FUNCTION_BLOCK PalletizerElevator EXTENDS Elevator
VAR_INPUT
END_VAR
VAR_OUTPUT
	isMoving : BOOL;
END_VAR
VAR
	fbElevatorMoving : Sensor;
	fbElevatorUp : BoolOut;
	fbElevatorDown : BoolOut;
	fbElevatorToLimit : BoolOut;
END_VAR

isMoving := fbElevatorMoving.bSignal;

PROPERTY getElevatorMoving : I_StepCondition
GET
getElevatorMoving := fbElevatorMoving.getSignal;
END_GET
END_PROPERTY

METHOD MoveDown : BOOL
VAR_INPUT
END_VAR
fbElevatorDown.setValue := TRUE;
fbElevatorUp.setValue := FALSE;

fbElevatorToLimit.setValue := TRUE;
END_METHOD

METHOD MoveUp : BOOL
VAR_INPUT
END_VAR
fbElevatorUp.setValue := TRUE;
fbElevatorDown.setValue := FALSE;

fbElevatorToLimit.setValue := TRUE;
END_METHOD

END_FUNCTION_BLOCK

(* stored: Version 1.1.0.1, ProductVersion 3.1.4024.2
   POU PalletizerElevator: Id {4eb779f8-64c2-45d2-8e33-ff6a6414ef2d}, SpecialFunc None
   Property getElevatorMoving: Id {95323b9c-95fa-41bd-8503-cd70b97b05a2}
   Get Get: Id {0e5bfb5b-cdd0-42ca-8764-48c3dad921a1}
   Method MoveDown: Id {f1df31ac-a5cc-42f8-8414-2af4b7cb61b7}
   Method MoveUp: Id {6365eaa9-072d-406d-bc17-1567ac647da2} *)
